Staubli VAL3: getTrajItem.pgx

public program getTrajItem(TrajectoryItem& x_tTraj[], num x_nIndex)
begin
  //
  // get all the FIELD
  //
  x_tTraj=pEditPoint.tData[x_nIndex].tSuper
end
